# EPICS autosave request: tests/testfiles/cfg/SF_QFF_PV.req
$(SYS):X
$(SYS):Y
